FUNCTION_BLOCK FlushingManagerSLB (* Basic Function Block Type *)
  (* Standard: 61499-2 *)
  (* Version 0.0, 8/23/2024, SESA713705, Schneider Electric, Template *)
  PACKAGE SE.Nereda;
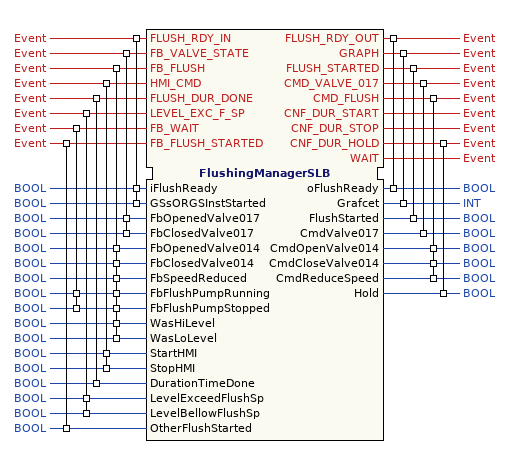
  EVENT_INPUT
    FLUSH_RDY_IN WITH iFlushReady, GSsORGSInstStarted;
    FB_VALVE_STATE WITH FbOpenedValve017, FbClosedValve017;
    FB_FLUSH WITH FbOpenedValve014, FbClosedValve014, FbSpeedReduced, FbFlushPumpRunning, FbFlushPumpStopped, WasHiLevel, WasLoLevel;
    HMI_CMD WITH StartHMI, StopHMI;
    FLUSH_DUR_DONE WITH DurationTimeDone;
    LEVEL_EXC_F_SP WITH LevelExceedFlushSp, LevelBellowFlushSp;
    FB_WAIT WITH FbFlushPumpRunning, FbFlushPumpStopped;
    FB_FLUSH_STARTED WITH OtherFlushStarted;
  END_EVENT
  EVENT_OUTPUT
    FLUSH_RDY_OUT WITH oFlushReady;
    GRAPH WITH Grafcet;
    FLUSH_STARTED WITH FlushStarted;
    CMD_VALVE_017 WITH CmdValve017;
    CMD_FLUSH WITH CmdOpenValve014, CmdCloseValve014, CmdReduceSpeed;
    CNF_DUR_START;
    CNF_DUR_STOP;
    CNF_DUR_HOLD WITH Hold;
    WAIT;
  END_EVENT
  VAR_INPUT
    iFlushReady : BOOL;
    GSsORGSInstStarted : BOOL;
    FbOpenedValve017 : BOOL;
    FbClosedValve017 : BOOL;
    FbOpenedValve014 : BOOL;
    FbClosedValve014 : BOOL;
    FbSpeedReduced : BOOL;
    FbFlushPumpRunning : BOOL;
    FbFlushPumpStopped : BOOL;
    WasHiLevel : BOOL;
    WasLoLevel : BOOL;
    StartHMI : BOOL;
    StopHMI : BOOL;
    DurationTimeDone : BOOL;
    LevelExceedFlushSp : BOOL;
    LevelBellowFlushSp : BOOL;
    OtherFlushStarted : BOOL;
  END_VAR
  VAR_OUTPUT
    oFlushReady : BOOL;
    Grafcet : INT;
    FlushStarted : BOOL;
    CmdValve017 : BOOL;
    CmdOpenValve014 : BOOL;
    CmdCloseValve014 : BOOL;
    CmdReduceSpeed : BOOL;
    Hold : BOOL;
  END_VAR
  EC_STATES
    START; (* Initial State *)
    START_FLUSH : OpenValve017 -> CMD_VALVE_017, -> GRAPH;
    START_DUR : FlushStarted -> CNF_DUR_START, -> FLUSH_STARTED, -> GRAPH;
    STOP_FLUSH : CloseValve017 -> CMD_VALVE_017, -> GRAPH;
    FLUSH_OFF : FlushOFF -> CNF_DUR_STOP, -> FLUSH_STARTED, -> FLUSH_RDY_OUT, -> CNF_DUR_HOLD, -> GRAPH;
    ReduceSpeed2 : ReduceSpeed -> CMD_FLUSH, -> GRAPH;
    CloseValve14 : CloseValve014 -> CMD_FLUSH, -> GRAPH;
    LevelExceedFlushSp;
    FlushRdy : FlushRdy -> FLUSH_RDY_OUT, -> GRAPH, -> CNF_DUR_HOLD;
    ReduceSpeed1 : ReduceSpeed -> CMD_FLUSH, -> GRAPH;
    OpenValve014_1 : OpenValve014 -> CMD_FLUSH, -> GRAPH, -> WAIT;
    CancelReduceSpeed : CancelReduceSpeed -> CMD_FLUSH, -> GRAPH;
    OpenValve014_2 : OpenValve014 -> CMD_FLUSH, -> GRAPH;
    CancelReduceSpeed1 : CancelReduceSpeed -> CMD_FLUSH, FlushingOff -> FLUSH_RDY_OUT, -> GRAPH;
    StopFlush;
    FlushingOFF : FlushingOff -> FLUSH_RDY_OUT;
    Hold : Hold -> CNF_DUR_HOLD, -> GRAPH;
  END_STATES
  EC_TRANSITIONS
    LevelExceedFlushSp TO FlushRdy := iFlushReady AND LevelBellowFlushSp AND NOT GSsORGSInstStarted;
    START_FLUSH TO CloseValve14 := FbOpenedValve017;
    START_DUR TO ReduceSpeed2 := DurationTimeDone OR NOT iFlushReady OR GSsORGSInstStarted;
    STOP_FLUSH TO CancelReduceSpeed1 := FbClosedValve017;
    FLUSH_OFF TO START := 1;
    OpenValve014_2 TO STOP_FLUSH := FbOpenedValve014 OR FbFlushPumpStopped OR OtherFlushStarted;
    CloseValve14 TO CancelReduceSpeed := FbClosedValve014;
    START TO LevelExceedFlushSp := LEVEL_EXC_F_SP AND LevelExceedFlushSp;
    START TO FlushRdy := HMI_CMD AND StartHMI AND NOT StopHMI;
    OpenValve014_1 TO ReduceSpeed1 := FbFlushPumpRunning;
    ReduceSpeed1 TO START_FLUSH := FbSpeedReduced;
    FlushRdy TO OpenValve014_1 := 1;
    CancelReduceSpeed TO START_DUR := NOT FbSpeedReduced;
    FlushingOFF TO OpenValve014_2 := WasHiLevel;
    CancelReduceSpeed1 TO FLUSH_OFF := (NOT FbSpeedReduced AND NOT iFlushReady) OR FbFlushPumpStopped;
    LevelExceedFlushSp TO FlushRdy := HMI_CMD AND StartHMI AND NOT StopHMI;
    OpenValve014_1 TO StopFlush := FB_WAIT AND FbFlushPumpStopped;
    ReduceSpeed1 TO StopFlush := FbFlushPumpStopped;
    START_FLUSH TO StopFlush := FbFlushPumpStopped;
    CloseValve14 TO StopFlush := FbFlushPumpStopped;
    CancelReduceSpeed TO StopFlush := FbFlushPumpStopped;
    START_DUR TO StopFlush := FbFlushPumpStopped;
    ReduceSpeed2 TO StopFlush := FbFlushPumpStopped;
    OpenValve014_2 TO StopFlush := FbFlushPumpStopped;
    StopFlush TO STOP_FLUSH := 1;
    FlushingOFF TO STOP_FLUSH := WasLoLevel OR FbFlushPumpStopped;
    ReduceSpeed2 TO FlushingOFF := FbSpeedReduced OR GSsORGSInstStarted;
    CancelReduceSpeed1 TO Hold := NOT FbSpeedReduced AND GSsORGSInstStarted;
    Hold TO FLUSH_OFF := NOT iFlushReady OR DurationTimeDone;
    Hold TO FlushRdy := NOT GSsORGSInstStarted AND iFlushReady AND NOT DurationTimeDone;
  END_TRANSITIONS
  ALGORITHM OpenValve017 IN ST:
;
Grafcet := 4;
CmdValve017 := TRUE;
  END_ALGORITHM
  ALGORITHM FlushStarted IN ST:
;
Grafcet := 7;
FlushStarted := TRUE;
  END_ALGORITHM
  ALGORITHM CloseValve017 IN ST:
;
Grafcet := 10;
CmdValve017 := FALSE;
  END_ALGORITHM
  ALGORITHM FlushOFF IN ST:
;
Grafcet := 12;
Hold := FALSE;
CmdValve017 := FALSE;
FlushStarted := FALSE;
oFlushReady := FALSE;
  END_ALGORITHM
  ALGORITHM OpenValve014 IN ST:
;
IF Grafcet = 1 THEN
	Grafcet := 2;
ELSIF Grafcet = 8 THEN
	Grafcet := 9;
END_IF;

CmdOpenValve014 := TRUE;
CmdCloseValve014 := FALSE;
  END_ALGORITHM
  ALGORITHM CancelReduceSpeed IN ST:
;
IF Grafcet = 5 THEN
	Grafcet := 6;
ELSIF Grafcet = 10 THEN
	Grafcet := 11;
END_IF;

CmdReduceSpeed := FALSE;
  END_ALGORITHM
  ALGORITHM FlushRdy IN ST:
;
Grafcet := 1;
Hold := FALSE;
IF StartHMI THEN
	oFlushReady := TRUE;
ELSE
	oFlushReady := iFlushReady;
END_IF;
  END_ALGORITHM
  ALGORITHM ReduceSpeed IN ST:
;
IF Grafcet = 2 THEN
	Grafcet := 3;
ELSIF Grafcet = 7 THEN
	Grafcet := 8;
END_IF;

CmdReduceSpeed := TRUE;
  END_ALGORITHM
  ALGORITHM CloseValve014 IN ST:
;
Grafcet := 5;
CmdOpenValve014 := FALSE;
CmdCloseValve014 := TRUE;
  END_ALGORITHM
  ALGORITHM FlushingOff IN ST:
;
oFlushReady := FALSE;
  END_ALGORITHM
  ALGORITHM Hold IN ST:
;
Hold := TRUE;
Grafcet := 13;
  END_ALGORITHM
END_FUNCTION_BLOCK
